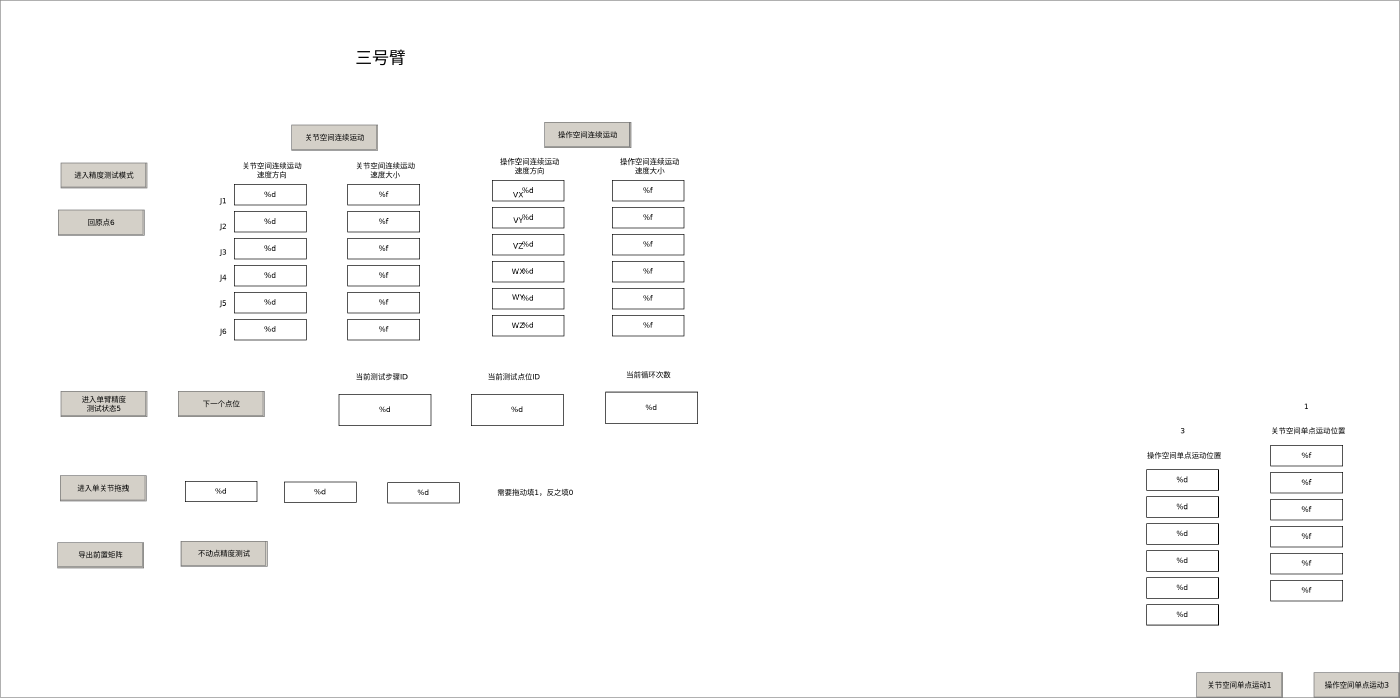
VISUALIZATION Robot_Jog_Arm3  // 2075x1035
    Button (90,241 128x38), "进入精度测试模式", colour toggle: GVL_AccuracyTestVar.g_enterPrecisionTestMode[3]
        toggle GVL_AccuracyTestVar.g_enterPrecisionTestMode[3]
    Label (489,64 150x43), "三号臂"
    Button (432,185 128x38), "关节空间连续运动", colour toggle: A1_Arm1ModeL[3,2]
        tap A1_Arm1Mode[3,2]
    Group (1773,997 302x38), invisible if: TRUE
        Button (174,0 128x38), "操作空间单点运动3", colour toggle: A1_Arm1ModeL[3,3]
            tap A1_Arm1Mode[3,3]
        Button (0,0 128x38), "关节空间单点运动1", colour toggle: A1_Arm1ModeL[3,1]
            tap A1_Arm1Mode[3,1]
    Button (807,181 128x38), "操作空间连续运动", colour toggle: A1_Arm1ModeL[3,4]
        tap A1_Arm1Mode[3,4]
    Button (86,311 128x38), "回原点6", colour toggle: A1_Arm1ModeL[3,6]
        tap A1_Arm1Mode[3,6]
    Rectangle (347,273 107x31), "%d", text variable: GVL_AccuracyTestVar.g_jntMotionDir[3][1]
        OnMouseClick: write the text variable via Default, min -1, max 1
    Label (328,238 150x29), "关节空间连续运动 速度方向"
    Rectangle (347,313 107x31), "%d", text variable: GVL_AccuracyTestVar.g_jntMotionDir[3][2]
        OnMouseClick: write the text variable via Default, min -1, max 1
    Rectangle (347,353 107x31), "%d", text variable: GVL_AccuracyTestVar.g_jntMotionDir[3][3]
        OnMouseClick: write the text variable via Default, min -1, max 1
    Rectangle (347,393 107x31), "%d", text variable: GVL_AccuracyTestVar.g_jntMotionDir[3][4]
        OnMouseClick: write the text variable via Default, min -1, max 1
    Rectangle (347,433 107x31), "%d", text variable: GVL_AccuracyTestVar.g_jntMotionDir[3][5]
        OnMouseClick: write the text variable via Default, min -1, max 1
    Rectangle (347,473 107x31), "%d", text variable: GVL_AccuracyTestVar.g_jntMotionDir[3][6]
        OnMouseClick: write the text variable via Default, min -1, max 1
    Group (1861,588 153x303), invisible if: TRUE
        Rectangle (22,72 107x31), "%f", text variable: GVL_AccuracyTestVar.g_targetJntPos[3][1]
            OnMouseClick: write the text variable via Default
        Label (3,36 150x30), "关节空间单点运动位置"
        Rectangle (22,112 107x31), "%f", text variable: GVL_AccuracyTestVar.g_targetJntPos[3][2]
            OnMouseClick: write the text variable via Default
        Rectangle (22,152 107x31), "%f", text variable: GVL_AccuracyTestVar.g_targetJntPos[3][3]
            OnMouseClick: write the text variable via Default
        Rectangle (22,192 107x31), "%f", text variable: GVL_AccuracyTestVar.g_targetJntPos[3][4]
            OnMouseClick: write the text variable via Default
        Rectangle (22,232 107x31), "%f", text variable: GVL_AccuracyTestVar.g_targetJntPos[3][5]
            OnMouseClick: write the text variable via Default
        Rectangle (22,272 107x31), "%f", text variable: GVL_AccuracyTestVar.g_targetJntPos[3][6]
            OnMouseClick: write the text variable via Default
        Label (0,0 150x30), "1"
    Rectangle (515,273 107x31), "%f", text variable: GVL_AccuracyTestVar.g_jntVel[3][1]
        OnMouseClick: write the text variable via Default
    Label (496,238 150x29), "关节空间连续运动 速度大小"
    Rectangle (515,313 107x31), "%f", text variable: GVL_AccuracyTestVar.g_jntVel[3][2]
        OnMouseClick: write the text variable via Default
    Rectangle (515,353 107x31), "%f", text variable: GVL_AccuracyTestVar.g_jntVel[3][3]
        OnMouseClick: write the text variable via Default
    Rectangle (515,393 107x31), "%f", text variable: GVL_AccuracyTestVar.g_jntVel[3][4]
        OnMouseClick: write the text variable via Default
    Rectangle (515,433 107x31), "%f", text variable: GVL_AccuracyTestVar.g_jntVel[3][5]
        OnMouseClick: write the text variable via Default
    Rectangle (515,473 107x31), "%f", text variable: GVL_AccuracyTestVar.g_jntVel[3][6]
        OnMouseClick: write the text variable via Default
    Group (1678,624 152x303), invisible if: TRUE
        Rectangle (21,72 107x31), "%d"
        Label (2,37 150x29), "操作空间单点运动位置"
        Rectangle (21,112 107x31), "%d"
        Rectangle (21,152 107x31), "%d"
        Rectangle (21,192 107x31), "%d"
        Rectangle (21,232 107x31), "%d"
        Rectangle (21,272 107x31), "%d"
        Label (0,0 150x30), "3"
    Rectangle (729,267 107x31), "%d", text variable: GVL_AccuracyTestVar.g_spatialMotionDir[3][1]
        OnMouseClick: write the text variable via Default, min -1, max 1
    Label (710,232 150x29), "操作空间连续运动 速度方向"
    Rectangle (729,307 107x31), "%d", text variable: GVL_AccuracyTestVar.g_spatialMotionDir[3][2]
        OnMouseClick: write the text variable via Default, min -1, max 1
    Rectangle (729,347 107x31), "%d", text variable: GVL_AccuracyTestVar.g_spatialMotionDir[3][3]
        OnMouseClick: write the text variable via Default, min -1, max 1
    Rectangle (729,387 107x31), "%d", text variable: GVL_AccuracyTestVar.g_spatialMotionDir[3][4]
        OnMouseClick: write the text variable via Default, min -1, max 1
    Rectangle (729,427 107x31), "%d", text variable: GVL_AccuracyTestVar.g_spatialMotionDir[3][5]
        OnMouseClick: write the text variable via Default, min -1, max 1
    Rectangle (729,467 107x31), "%d", text variable: GVL_AccuracyTestVar.g_spatialMotionDir[3][6]
        OnMouseClick: write the text variable via Default, min -1, max 1
    Rectangle (907,267 107x31), "%f", text variable: GVL_AccuracyTestVar.g_spatialVel[3][1]
        OnMouseClick: write the text variable via Default
    Label (888,232 150x29), "操作空间连续运动 速度大小"
    Rectangle (907,307 107x31), "%f", text variable: GVL_AccuracyTestVar.g_spatialVel[3][2]
        OnMouseClick: write the text variable via Default
    Rectangle (907,347 107x31), "%f", text variable: GVL_AccuracyTestVar.g_spatialVel[3][3]
        OnMouseClick: write the text variable via Default
    Rectangle (907,387 107x31), "%f", text variable: GVL_AccuracyTestVar.g_spatialVel[3][4]
        OnMouseClick: write the text variable via Default
    Rectangle (907,427 107x31), "%f", text variable: GVL_AccuracyTestVar.g_spatialVel[3][5]
        OnMouseClick: write the text variable via Default
    Rectangle (907,467 107x31), "%f", text variable: GVL_AccuracyTestVar.g_spatialVel[3][6]
        OnMouseClick: write the text variable via Default
    Button (90,580 128x38), "进入单臂精度 测试状态5", colour toggle: A1_Arm1ModeL[3,5]
        toggle A1_Arm1Mode[3,5]
    Button (264,580 128x38), "下一个点位", colour toggle: GVL_AccuracyTestVar.g_nextStep[2]
        tap GVL_AccuracyTestVar.g_nextStep[3]
    Group (491,541 545x90)
        Rectangle (11,43 137x47), "%d", text variable: GVL_AccuracyTestVar.g_curStep[3]
        Label (0,3 150x30), "当前测试步骤ID"
        Rectangle (207,43 137x47), "%d", text variable: GVL_AccuracyTestVar.g_testPointId[3]
        Label (196,3 150x30), "当前测试点位ID"
        Rectangle (406,40 137x47), "%d", text variable: GVL_AccuracyTestVar.g_testCycleId[3]
        Label (395,0 150x30), "当前循环次数"
    Group (324,283 14x224)
        Label (0,0 14x30), "J1"
        Label (0,38 14x30), "J2"
        Label (0,76 14x30), "J3"
        Label (0,114 14x30), "J4"
        Label (0,152 14x30), "J5"
        Label (0,194 14x30), "J6"
    Group (693,274 26x224)
        Label (0,0 150x30), "VX"
        Label (0,38 150x30), "VY"
        Label (0,76 150x30), "VZ"
        Label (0,114 150x30), "WX"
        Label (0,152 150x30), "WY"
        Label (0,194 150x30), "WZ"
    Rectangle (274,713 107x31), "%d", text variable: GVL_AccuracyTestVar.g_dragJntFlag[3][1]
        OnMouseClick: write the text variable via Default, min -1, max 1
    Button (89,705 128x38), "进入单关节拖拽", colour toggle: A1_Arm1ModeL[3,7]
        toggle A1_Arm1Mode[3,7]
    Rectangle (421,714 107x31), "%d", text variable: GVL_AccuracyTestVar.g_dragJntFlag[3][2]
        OnMouseClick: write the text variable via Default, min -1, max 1
    Rectangle (574,715 107x31), "%d", text variable: GVL_AccuracyTestVar.g_dragJntFlag[3][3]
        OnMouseClick: write the text variable via Default, min -1, max 1
    Label (710,716 167x29), "需要拖动填1，反之填0"
    Button (85,804 128x38), "导出前置矩阵"
        tap GVL_AccuracyTestVar.g_writeData[3]
    Button (268,802 128x38), "不动点精度测试", colour toggle: A1_Arm1ModeL[1,5]
        toggle A1_Arm1Mode[3,8]
END_VISUALIZATION

(* stored: Version 1.1.0.1, ProductVersion 3.1.4024.11
   Visu Robot_Jog_Arm3: Id {cba8aa8c-b6b5-405f-a7d8-cd0d47d13066} *)
